INTERFACE I_SnappyConfig EXTENDS I_SnappySetup, I_SnappySetupConfigBuild

PROPERTY bIsConfigured : BOOL
GET
END_GET
END_PROPERTY

PROPERTY itfRpcProxy : I_RpcProxy
GET
END_GET
END_PROPERTY

PROPERTY itfSerializer : I_Serializer
GET
END_GET
END_PROPERTY

PROPERTY itfTestFramework : I_TestFrameWorkAdapter
GET
END_GET
END_PROPERTY

END_INTERFACE

(* stored: Version 1.1.0.1, ProductVersion 3.1.4026.18
   Itf I_SnappyConfig: Id {63677510-8b39-4b00-b887-d436bf424311}
   Property bIsConfigured: Id {a8912a0c-d11f-4856-9e0a-01170623bfed}
   Get Get: Id {216dd96f-3194-44d6-af01-f658a880d89f}
   Property itfRpcProxy: Id {5d200fb7-94a2-4950-bf6e-ee9a81561722}
   Get Get: Id {201a5c86-084a-448b-b263-0b4e24458780}
   Property itfSerializer: Id {07aa9712-80a0-4c37-81ec-37706ac84604}
   Get Get: Id {582174c1-76e4-4007-ac8d-c8fe94a1d98c}
   Property itfTestFramework: Id {6cf81d96-7267-4fbd-89a0-99fce29166e8}
   Get Get: Id {c1c48e0d-f791-42e3-85c7-a8bee555e35b} *)
